TYPE ST_PU_Stellwert :
STRUCT
	Betrieb			: BOOL;

	Leistung		: USINT;
END_STRUCT
END_TYPE

(* stored: Version 1.1.0.1, ProductVersion 3.1.4024.9
   DUT ST_PU_Stellwert: Id {73b3cd4e-8894-4c2d-88f8-385e0e576122} *)
